(* IEC 61131-3 sources: Daniele1996.github.io/AUTOMATION_AND_SOFTWARE_DESIGN_PATTERN/AUTOMATION_STUDIO/Task1/Logical/OSP, 5 files *)

(* ---- Types.typ ---- *)
TYPE

END_TYPE

(* ---- Cyclic.st ---- *)
PROGRAM _CYCLIC
	(* Insert code here *)

	IF Machine_Handler.Run THEN
		Led_Start := TRUE;
		Led_Stop := TRUE;

	ELSIF NOT Machine_Handler.Run AND NOT Machine_Handler.Initialize AND Init_logical AND NOT Machine_Handler.On_Phase_Stop THEN
		Blink(LED := Led_Start);
		Led_Stop := FALSE;

	ELSE
		Led_Start := FALSE;
		Led_Stop := FALSE;

	END_IF;

END_PROGRAM

(* ---- Exit.st ---- *)
PROGRAM _EXIT
	(* Insert code here *)

END_PROGRAM

(* ---- Init.st ---- *)
PROGRAM _INIT
	(* Insert code here *)

END_PROGRAM

(* ---- Variables.var ---- *)
VAR
	Led_Start : BOOL;
	Led_Stop : BOOL;
	Led_Reset : BOOL;
	Blink : BlinkFB;
END_VAR
